FUNCTION_BLOCK SS5 (* Composite FB wrapping other FBs *)
  (* Standard: 61499-2 *)
  (* Version 1.0, 2024-10-03, DEVIASH *)
  PACKAGE UserLibs::SubStations::SS5;
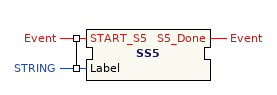
  EVENT_INPUT
    START_S5 WITH Label; (* Initialization Request *)
  END_EVENT
  EVENT_OUTPUT
    S5_Done; (* Initialization Confirm *)
  END_EVENT
  VAR_INPUT
    Label : STRING;
  END_VAR
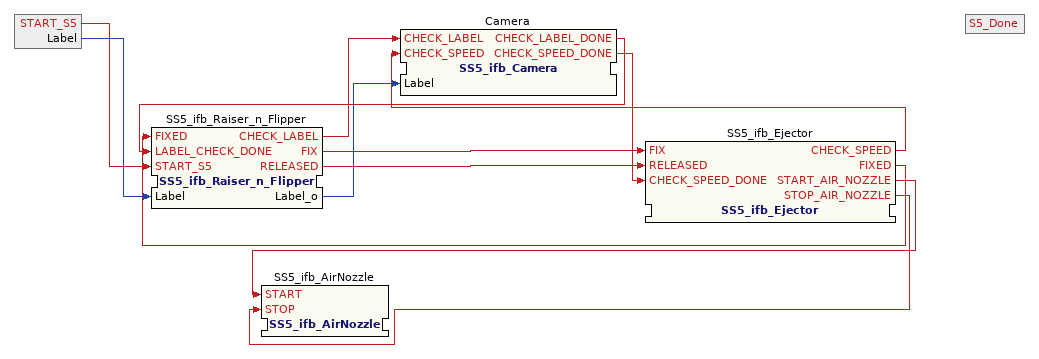
  FBS
    Camera : UserLibs::SubStations::SS5::SS5_ifb_Camera;
    SS5_ifb_AirNozzle : SS5_ifb_AirNozzle;
    SS5_ifb_Ejector : UserLibs::SubStations::SS5::SS5_ifb_Ejector;
    SS5_ifb_Raiser_n_Flipper : UserLibs::SubStations::SS5::SS5_ifb_Raiser_n_Flipper;
  END_FBS
  EVENT_CONNECTIONS
    SS5_ifb_Raiser_n_Flipper.CHECK_LABEL TO Camera.CHECK_LABEL;
    SS5_ifb_Ejector.CHECK_SPEED TO Camera.CHECK_SPEED;
    SS5_ifb_Ejector.FIXED TO SS5_ifb_Raiser_n_Flipper.FIXED;
    SS5_ifb_Raiser_n_Flipper.FIX TO SS5_ifb_Ejector.FIX;
    SS5_ifb_Raiser_n_Flipper.RELEASED TO SS5_ifb_Ejector.RELEASED;
    SS5_ifb_Ejector.START_AIR_NOZZLE TO SS5_ifb_AirNozzle.START;
    SS5_ifb_Ejector.STOP_AIR_NOZZLE TO SS5_ifb_AirNozzle.STOP;
    Camera.CHECK_LABEL_DONE TO SS5_ifb_Raiser_n_Flipper.LABEL_CHECK_DONE;
    Camera.CHECK_SPEED_DONE TO SS5_ifb_Ejector.CHECK_SPEED_DONE;
    START_S5 TO SS5_ifb_Raiser_n_Flipper.START_S5;
  END_CONNECTIONS
  DATA_CONNECTIONS
    SS5_ifb_Raiser_n_Flipper.Label_o TO Camera.Label;
    Label TO SS5_ifb_Raiser_n_Flipper.Label;
  END_CONNECTIONS
END_FUNCTION_BLOCK
